DATA_BLOCK "Data_block_1"
{ S7_Optimized_Access := 'TRUE' }
VERSION : 0.1
NON_RETAIN
   VAR
      Etat : Array[0..235] of DInt;
      Action : Array[0..235] of Int;
   END_VAR
BEGIN
   Etat[0] := 0;
   Etat[1] := 3528021;
   Etat[2] := 5592151;
   Etat[3] := 5592407;
   Etat[4] := 5594613;
   Etat[5] := 5594869;
   Etat[6] := 5723477;
   Etat[7] := 6116693;
   Etat[8] := 7705941;
   Etat[9] := 7722325;
   Etat[10] := 9789141;
   Etat[11] := 9789397;
   Etat[12] := 9794901;
   Etat[13] := 9917781;
   Etat[14] := 10310997;
   Etat[15] := 11883605;
   Etat[16] := 11883861;
   Etat[17] := 13976661;
   Etat[18] := 13988949;
   Etat[19] := 13989205;
   Etat[20] := 14112085;
   Etat[21] := 16078165;
   Etat[22] := 18174805;
   Etat[23] := 18175069;
   Etat[24] := 18175325;
   Etat[25] := 18177525;
   Etat[26] := 18183509;
   Etat[27] := 18306389;
   Etat[28] := 19256661;
   Etat[29] := 20305237;
   Etat[30] := 20305493;
   Etat[31] := 21321045;
   Etat[32] := 22304085;
   Etat[33] := 22304597;
   Etat[34] := 22306805;
   Etat[35] := 22353237;
   Etat[36] := 22368341;
   Etat[37] := 22368343;
   Etat[38] := 22369109;
   Etat[39] := 22369111;
   Etat[40] := 22369301;
   Etat[41] := 22369349;
   Etat[42] := 22369361;
   Etat[43] := 22369364;
   Etat[44] := 22369367;
   Etat[45] := 22369373;
   Etat[46] := 22369617;
   Etat[47] := 22369620;
   Etat[48] := 22369623;
   Etat[49] := 22369629;
   Etat[50] := 22369813;
   Etat[51] := 22369879;
   Etat[52] := 22369885;
   Etat[53] := 22370069;
   Etat[54] := 22370117;
   Etat[55] := 22370129;
   Etat[56] := 22370135;
   Etat[57] := 22370141;
   Etat[58] := 22370805;
   Etat[59] := 22371317;
   Etat[60] := 22371573;
   Etat[61] := 22371813;
   Etat[62] := 22371829;
   Etat[63] := 22372085;
   Etat[64] := 22372277;
   Etat[65] := 22372325;
   Etat[66] := 22372341;
   Etat[67] := 22373717;
   Etat[68] := 22377813;
   Etat[69] := 22500693;
   Etat[70] := 22631765;
   Etat[71] := 23450965;
   Etat[72] := 23451221;
   Etat[73] := 24483157;
   Etat[74] := 24499285;
   Etat[75] := 24499541;
   Etat[76] := 25515349;
   Etat[77] := 25515861;
   Etat[78] := 26498389;
   Etat[79] := 26498901;
   Etat[80] := 26501077;
   Etat[81] := 26559829;
   Etat[82] := 26562645;
   Etat[83] := 26563413;
   Etat[84] := 26563677;
   Etat[85] := 26563921;
   Etat[86] := 26563933;
   Etat[87] := 26564189;
   Etat[88] := 26564373;
   Etat[89] := 26564433;
   Etat[90] := 26564445;
   Etat[91] := 26565333;
   Etat[92] := 26565589;
   Etat[93] := 26565845;
   Etat[94] := 26566101;
   Etat[95] := 26566357;
   Etat[96] := 26566549;
   Etat[97] := 26566613;
   Etat[98] := 26568021;
   Etat[99] := 26571861;
   Etat[100] := 26572117;
   Etat[101] := 26694741;
   Etat[102] := 26694997;
   Etat[103] := 26826069;
   Etat[104] := 27612245;
   Etat[105] := 27612501;
   Etat[106] := 27613013;
   Etat[107] := 28660821;
   Etat[108] := 28661077;
   Etat[109] := 28661333;
   Etat[110] := 28661589;
   Etat[111] := 29709653;
   Etat[112] := 30692693;
   Etat[113] := 30693205;
   Etat[114] := 30695381;
   Etat[115] := 30753877;
   Etat[116] := 30754133;
   Etat[117] := 30756949;
   Etat[118] := 30757461;
   Etat[119] := 30758225;
   Etat[120] := 30758228;
   Etat[121] := 30758237;
   Etat[122] := 30759637;
   Etat[123] := 30760661;
   Etat[124] := 30760917;
   Etat[125] := 30762069;
   Etat[126] := 30762325;
   Etat[127] := 30766165;
   Etat[128] := 30766421;
   Etat[129] := 30889045;
   Etat[130] := 30889301;
   Etat[131] := 31806805;
   Etat[132] := 32855125;
   Etat[133] := 32855381;
   Etat[134] := 34954869;
   Etat[135] := 34955125;
   Etat[136] := 34985045;
   Etat[137] := 34985301;
   Etat[138] := 35083605;
   Etat[139] := 35476821;
   Etat[140] := 38884693;
   Etat[141] := 39081301;
   Etat[142] := 39081813;
   Etat[143] := 39083893;
   Etat[144] := 39145557;
   Etat[145] := 39145559;
   Etat[146] := 39146325;
   Etat[147] := 39146327;
   Etat[148] := 39146583;
   Etat[149] := 39146836;
   Etat[150] := 39146839;
   Etat[151] := 39148405;
   Etat[152] := 39148661;
   Etat[153] := 39148917;
   Etat[154] := 39149157;
   Etat[155] := 39149173;
   Etat[156] := 39149413;
   Etat[157] := 39149429;
   Etat[158] := 39163221;
   Etat[159] := 39179349;
   Etat[160] := 39179605;
   Etat[161] := 39179861;
   Etat[162] := 39277653;
   Etat[163] := 39277909;
   Etat[164] := 39408981;
   Etat[165] := 39670869;
   Etat[166] := 39671125;
   Etat[167] := 43078997;
   Etat[168] := 43337045;
   Etat[169] := 43340629;
   Etat[170] := 43340885;
   Etat[171] := 43341141;
   Etat[172] := 43341653;
   Etat[173] := 43342677;
   Etat[174] := 43342933;
   Etat[175] := 43343189;
   Etat[176] := 43343445;
   Etat[177] := 43343701;
   Etat[178] := 43349077;
   Etat[179] := 43349333;
   Etat[180] := 43471957;
   Etat[181] := 43472213;
   Etat[182] := 43865173;
   Etat[183] := 43865429;
   Etat[184] := 47469909;
   Etat[185] := 47470421;
   Etat[186] := 47472469;
   Etat[187] := 47531093;
   Etat[188] := 47531349;
   Etat[189] := 47535444;
   Etat[190] := 47535445;
   Etat[191] := 47537749;
   Etat[192] := 47538005;
   Etat[193] := 47539285;
   Etat[194] := 47539541;
   Etat[195] := 47543381;
   Etat[196] := 47543637;
   Etat[197] := 47666517;
   Etat[198] := 51762517;
   Etat[199] := 51860821;
   Etat[200] := 51991893;
   Etat[201] := 52253781;
   Etat[202] := 52254037;
   Etat[203] := 55661653;
   Etat[204] := 55661909;
   Etat[205] := 55858517;
   Etat[206] := 55907669;
   Etat[207] := 55923793;
   Etat[208] := 55924049;
   Etat[209] := 55924055;
   Etat[210] := 55940437;
   Etat[211] := 55956821;
   Etat[212] := 56055125;
   Etat[213] := 56185941;
   Etat[214] := 56186197;
   Etat[215] := 56448085;
   Etat[216] := 56448341;
   Etat[217] := 59855957;
   Etat[218] := 59856213;
   Etat[219] := 60052821;
   Etat[220] := 60053333;
   Etat[221] := 60055381;
   Etat[222] := 60118353;
   Etat[223] := 60118357;
   Etat[224] := 60118865;
   Etat[225] := 60120917;
   Etat[226] := 60249173;
   Etat[227] := 60249429;
   Etat[228] := 60380245;
   Etat[229] := 60380501;
   Etat[230] := 60642389;
   Etat[231] := 60642645;
   Etat[232] := 60642901;
   Etat[233] := 60643153;
   Etat[234] := 64312661;
   Etat[235] := 67108865;
   Action[0] := 2;
   Action[1] := 0;
   Action[2] := 13;
   Action[3] := 13;
   Action[4] := 11;
   Action[5] := 0;
   Action[6] := 5;
   Action[7] := 4;
   Action[8] := 0;
   Action[9] := 3;
   Action[10] := 8;
   Action[11] := 10;
   Action[12] := 7;
   Action[13] := 5;
   Action[14] := 4;
   Action[15] := 3;
   Action[16] := 3;
   Action[17] := 0;
   Action[18] := 2;
   Action[19] := 7;
   Action[20] := 5;
   Action[21] := 3;
   Action[22] := 0;
   Action[23] := 12;
   Action[24] := 12;
   Action[25] := 8;
   Action[26] := 7;
   Action[27] := 5;
   Action[28] := 0;
   Action[29] := 6;
   Action[30] := 3;
   Action[31] := 0;
   Action[32] := 0;
   Action[33] := 0;
   Action[34] := 0;
   Action[35] := 0;
   Action[36] := 0;
   Action[37] := 0;
   Action[38] := 9;
   Action[39] := 9;
   Action[40] := 0;
   Action[41] := 0;
   Action[42] := 0;
   Action[43] := 0;
   Action[44] := 13;
   Action[45] := 12;
   Action[46] := 0;
   Action[47] := 0;
   Action[48] := 13;
   Action[49] := 12;
   Action[50] := 0;
   Action[51] := 0;
   Action[52] := 0;
   Action[53] := 9;
   Action[54] := 9;
   Action[55] := 9;
   Action[56] := 9;
   Action[57] := 12;
   Action[58] := 0;
   Action[59] := 9;
   Action[60] := 11;
   Action[61] := 0;
   Action[62] := 8;
   Action[63] := 11;
   Action[64] := 9;
   Action[65] := 9;
   Action[66] := 9;
   Action[67] := 0;
   Action[68] := 7;
   Action[69] := 5;
   Action[70] := 0;
   Action[71] := 0;
   Action[72] := 0;
   Action[73] := 0;
   Action[74] := 6;
   Action[75] := 3;
   Action[76] := 0;
   Action[77] := 9;
   Action[78] := 0;
   Action[79] := 0;
   Action[80] := 0;
   Action[81] := 0;
   Action[82] := 0;
   Action[83] := 0;
   Action[84] := 12;
   Action[85] := 0;
   Action[86] := 12;
   Action[87] := 12;
   Action[88] := 9;
   Action[89] := 0;
   Action[90] := 9;
   Action[91] := 0;
   Action[92] := 9;
   Action[93] := 10;
   Action[94] := 8;
   Action[95] := 10;
   Action[96] := 9;
   Action[97] := 9;
   Action[98] := 0;
   Action[99] := 7;
   Action[100] := 7;
   Action[101] := 0;
   Action[102] := 5;
   Action[103] := 0;
   Action[104] := 0;
   Action[105] := 0;
   Action[106] := 0;
   Action[107] := 3;
   Action[108] := 3;
   Action[109] := 3;
   Action[110] := 9;
   Action[111] := 2;
   Action[112] := 2;
   Action[113] := 2;
   Action[114] := 2;
   Action[115] := 2;
   Action[116] := 0;
   Action[117] := 0;
   Action[118] := 0;
   Action[119] := 2;
   Action[120] := 0;
   Action[121] := 12;
   Action[122] := 0;
   Action[123] := 8;
   Action[124] := 9;
   Action[125] := 2;
   Action[126] := 2;
   Action[127] := 7;
   Action[128] := 7;
   Action[129] := 2;
   Action[130] := 5;
   Action[131] := 0;
   Action[132] := 0;
   Action[133] := 2;
   Action[134] := 11;
   Action[135] := 11;
   Action[136] := 0;
   Action[137] := 6;
   Action[138] := 0;
   Action[139] := 4;
   Action[140] := 0;
   Action[141] := 0;
   Action[142] := 0;
   Action[143] := 0;
   Action[144] := 0;
   Action[145] := 0;
   Action[146] := 9;
   Action[147] := 9;
   Action[148] := 13;
   Action[149] := 0;
   Action[150] := 13;
   Action[151] := 9;
   Action[152] := 11;
   Action[153] := 0;
   Action[154] := 0;
   Action[155] := 11;
   Action[156] := 9;
   Action[157] := 9;
   Action[158] := 0;
   Action[159] := 6;
   Action[160] := 6;
   Action[161] := 0;
   Action[162] := 0;
   Action[163] := 5;
   Action[164] := 0;
   Action[165] := 4;
   Action[166] := 4;
   Action[167] := 0;
   Action[168] := 0;
   Action[169] := 9;
   Action[170] := 0;
   Action[171] := 0;
   Action[172] := 9;
   Action[173] := 9;
   Action[174] := 0;
   Action[175] := 8;
   Action[176] := 8;
   Action[177] := 9;
   Action[178] := 7;
   Action[179] := 7;
   Action[180] := 0;
   Action[181] := 5;
   Action[182] := 0;
   Action[183] := 4;
   Action[184] := 0;
   Action[185] := 2;
   Action[186] := 0;
   Action[187] := 2;
   Action[188] := 2;
   Action[189] := 0;
   Action[190] := 2;
   Action[191] := 2;
   Action[192] := 9;
   Action[193] := 2;
   Action[194] := 2;
   Action[195] := 7;
   Action[196] := 7;
   Action[197] := 5;
   Action[198] := 1;
   Action[199] := 1;
   Action[200] := 0;
   Action[201] := 4;
   Action[202] := 1;
   Action[203] := 1;
   Action[204] := 1;
   Action[205] := 1;
   Action[206] := 0;
   Action[207] := 0;
   Action[208] := 0;
   Action[209] := 1;
   Action[210] := 1;
   Action[211] := 1;
   Action[212] := 5;
   Action[213] := 1;
   Action[214] := 1;
   Action[215] := 1;
   Action[216] := 4;
   Action[217] := 1;
   Action[218] := 1;
   Action[219] := 1;
   Action[220] := 1;
   Action[221] := 0;
   Action[222] := 0;
   Action[223] := 1;
   Action[224] := 0;
   Action[225] := 1;
   Action[226] := 0;
   Action[227] := 5;
   Action[228] := 1;
   Action[229] := 1;
   Action[230] := 4;
   Action[231] := 4;
   Action[232] := 0;
   Action[233] := 9;
   Action[234] := 2;
   Action[235] := 0;
END_DATA_BLOCK